FUNCTION_BLOCK FB_BPRequestor
VAR_INPUT
	stReqBP	:	ST_BeamParams;
END_VAR
VAR_OUTPUT
	q_stReqBP :	ST_BeamParams;
	q_ReqAtt  : REAL;
END_VAR
VAR
	
END_VAR

q_stReqBP := stReqBP;
q_ReqAtt := stReqBP.fAtt;

END_FUNCTION_BLOCK

(* stored: Version 1.1.0.1, ProductVersion 3.1.4024.0
   POU FB_BPRequestor: Id {936fd650-d613-49d0-b979-ce2a79a2ad53}, SpecialFunc None *)
